ABB RobotStudio station: 20204 CCSU ROS EGM_20240522-114910.rsstn

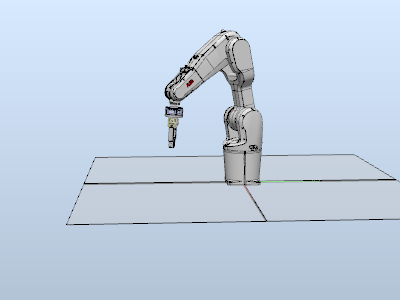
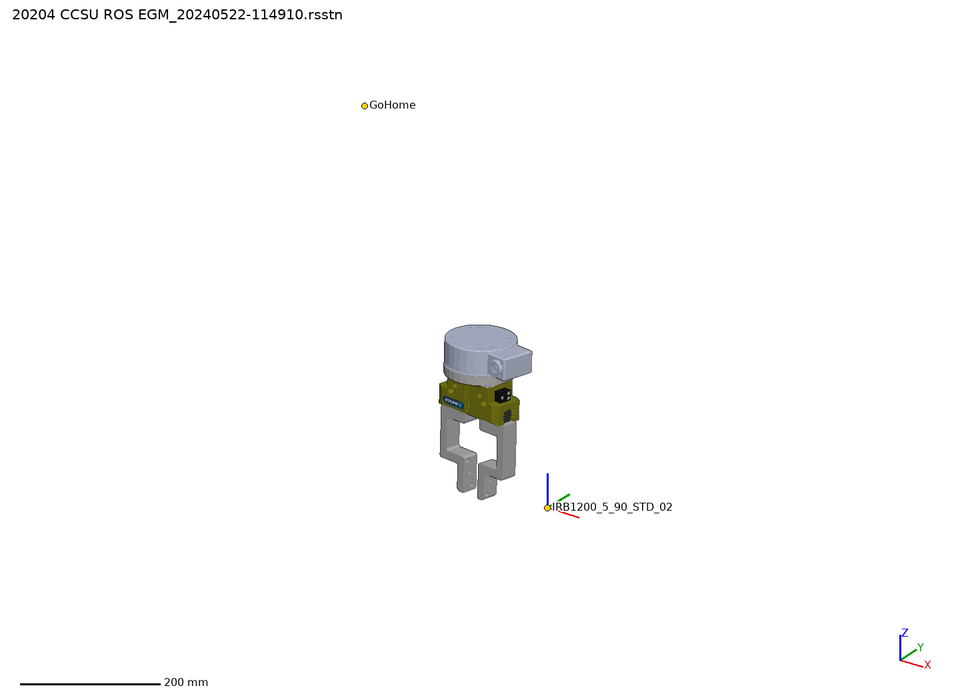
[picture v1: parts stored in the station drawn from their meshes, with robot base, taught points and paths (robot models come from the ABB library and are not in the file)]
Station 20204 CCSU RS (saved by RobotStudio 22.3.10098.0)
Controller 1200-800743_OfflineStation
  mechanical unit ROB_1: IRB1200_5_90_STD_02, 6 joints, base frame (0, 0, 0) mm
Layout (positions relative to the parent item):
  - IRB1200_5_90_STD_02 [mechanism, from %ABB.RobotStudio.Models.IRB1200%\IRB1200_5_90_STD_03.rslib] at (0, 0, 0) mm; joint values [-1.1589, 0.2025, 0.4737, -0.0167, 0.8192, 0.5941] (rad or m)
  - GRIPPER ONLY [part] at (189, -435.06, 506.71) mm, rotated rx 176.01 ry -1.8 rz -9.75 deg, size 125.6 x 50 x 198.4 mm
  - GRIPPER FORCE SENSOR [part] at (189, -435.06, 506.71) mm, rotated rx 176.01 ry -1.8 rz -9.75 deg, size 142.7 x 104 x 238.4 mm
Attachment: GRIPPER ONLY is attached to IRB1200_5_90_STD_02 / Link6
Attachment: GRIPPER FORCE SENSOR is attached to IRB1200_5_90_STD_02 / Link6
Targets, tools, work objects and paths stored in the station, written as RAPID:
! task T_ROB1
MODULE FORCENewProgram
  CONST robtarget GoHome:=[[-163.21,-220.75,679.83],[0.000017864,-0.460993,0.887404,0.000003505],[-2,0,1,0],[9E+09,9E+09,9E+09,9E+09,9E+09,9E+09]];
  PROC Main()
    rGoHome;
  ENDPROC
  PROC rGoHome()
    MoveJ GoHome,v500,z50,tool0;
  ENDPROC
ENDMODULE

! task T_ROB1
MODULE FORCECONTROL
  PROC FCRefStop()
  ENDPROC
  PROC FCRefStart()
  ENDPROC
  PROC FCDeact()
  ENDPROC
  PROC FCResetDampTune()
  ENDPROC
  PROC FCWaitNoRobMot()
  ENDPROC
ENDMODULE

! task T_ROB1
MODULE FCMACHINING
  PROC FCSpdChgDeact()
  ENDPROC
ENDMODULE

! task T_ROB1
MODULE user
  TASK PERS tooldata Gripper:=[TRUE,[[0,0,170],[1,0,0,0]],[1,[0,0,1],[1,0,0,0],0,0,0]];
  TASK PERS tooldata Gripper_FS:=[TRUE,[[0,0,225],[1,0,0,0]],[4,[-2.2,4.3,81.2],[1,0,0,0],0,0,0.006]];
ENDMODULE

! task T_ROB1
MODULE Tooling
  PROC rStopRunAtiTool()
    SetDO DOAtiSpindleStartSMC4,0;
    WaitTime \InPos,40;
    SetDO DOAtiSpindleCompSMC6,0;
  ENDPROC
  PROC rGripperOpen()
    SetDO DOGripperCloseSMC0,0;
    SetDO DOGripperOpenSMC2,1;
  ENDPROC
  PROC rGripperClose()
    SetDO DOGripperOpenSMC2,0;
    SetDO DOGripperCloseSMC0,1;
  ENDPROC
  PROC rRunAtiTool()
    SetDO DOAtiSpindleCompSMC6,1;
    WaitTime \InPos,1;
    SetDO DOAtiSpindleStartSMC4,1;
  ENDPROC
ENDMODULE

